// TIA Portal project "2022.05.31_第四章_移动指令3" (V17)

(* hardware
DEVICE "S7-1500/ET200MP station_1"  S7-1500 station
   slot 0: "导轨_0"  Rack  6ES7 590-1***0-0AA0
   slot 1: "PLC_1500"  CPU 1516-3 PN/DP  6ES7 516-3AN00-0AB0  V1.7
      slot 3: "CPU 显示_1"  6ES7591-1BA00-0AA0
      slot 32768: "PROFINET 接口_1"  X1
         slot 32769: "端口_1"  X1 P1
         slot 32770: "端口_2"  X1 P2
      slot 33024: "PROFINET 接口_2"  X2
         slot 33025: "端口_1"  X2 P1
      slot 33280: "DP 接口_1"  X3
DEVICE "HMI_1"  TP1200 Comfort
   slot 0: "HMI_1"  TP1200 Comfort  6AV2 124-0MC01-0AX0  17.0.0.0
   slot 1: "HMI_RT_1"  TP1200 Comfort  6AV2 124-0MC01-0AX0  17.0.0.0
   slot 5: "HMI_1.IE_CP_1"  PROFINET Interface  17.0.0.0
      slot 1: "PROFINET Interface_1"  PROFINET Interface
         slot 1: "Port_1"  Port
         slot 2: "Port_2"  Port
   slot 7: "HMI_1.MPI/DP_CP_1"  MPI/DP Interface  17.0.0.0
*)

// ===== PLC "PLC_1500"  CPU 1516-3 PN/DP =====

DATA_BLOCK "DATE_AND_TIME"   // DB1
{ S7_Optimized_Access := 'TRUE' }
VERSION : 0.1
   VAR
      "time" : Date_And_Time;
      time_ret : Int;
   END_VAR
BEGIN
END_DATA_BLOCK

DATA_BLOCK "启动操作DB"   // DB3
{ S7_Optimized_Access := 'TRUE' }
VERSION : 0.1
   VAR
      从数据数据块中读取按钮 : Bool;
      RET_VAL : Word;
      VALUE : Int;
      写入Array数据块 : Struct
         写入 : Bool;
         按钮 : Bool;
         RET_VAl : Word;
         VALUE : Int;
         写入装载存储器Array数据读取 : Struct
            按钮 : Bool;
            开始读取 : Bool;
            BUSY : Bool;
            DONE : Bool;
            error : Word;
            VALUE : Int;
            写入 : Bool;
            从装载存储器读取Array数据块 : Struct
               按钮 : Bool;
               读取 : Bool;
               BUSY : Bool;
               value : Int;
               done : Bool;
               error : Word;
            END_STRUCT;
         END_STRUCT;
      END_STRUCT;
   END_VAR
BEGIN
END_DATA_BLOCK

DATA_BLOCK "数组数据块A"   // DB4
{ S7_Optimized_Access := 'TRUE' }
VERSION : 0.1
   VAR
      Header : ArrayDBHeader;
      THIS : Array[0..10] of Int;
   END_VAR
BEGIN
END_DATA_BLOCK

DATA_BLOCK "装载数据块"   // DB5
{ S7_Optimized_Access := 'TRUE' }
VERSION : 0.1
BEGIN
END_DATA_BLOCK

FUNCTION_BLOCK "移动指令"   // FB1, LAD
{ S7_Optimized_Access := 'TRUE' }
VERSION : 0.1
   VAR
      ReadFromArrayDBL_Instance : ReadFromArrayDBL;
      WriteToArrayDBL_Instance : WriteToArrayDBL;
      IEC_Timer_0_Instance : TON_TIME;
   END_VAR
   VAR_TEMP   // added for the SCL form of the ladder/FBD networks
      _w1 : Bool;
   END_VAR
BEGIN

REGION Network 1: 从装载存储器Array的数据模块
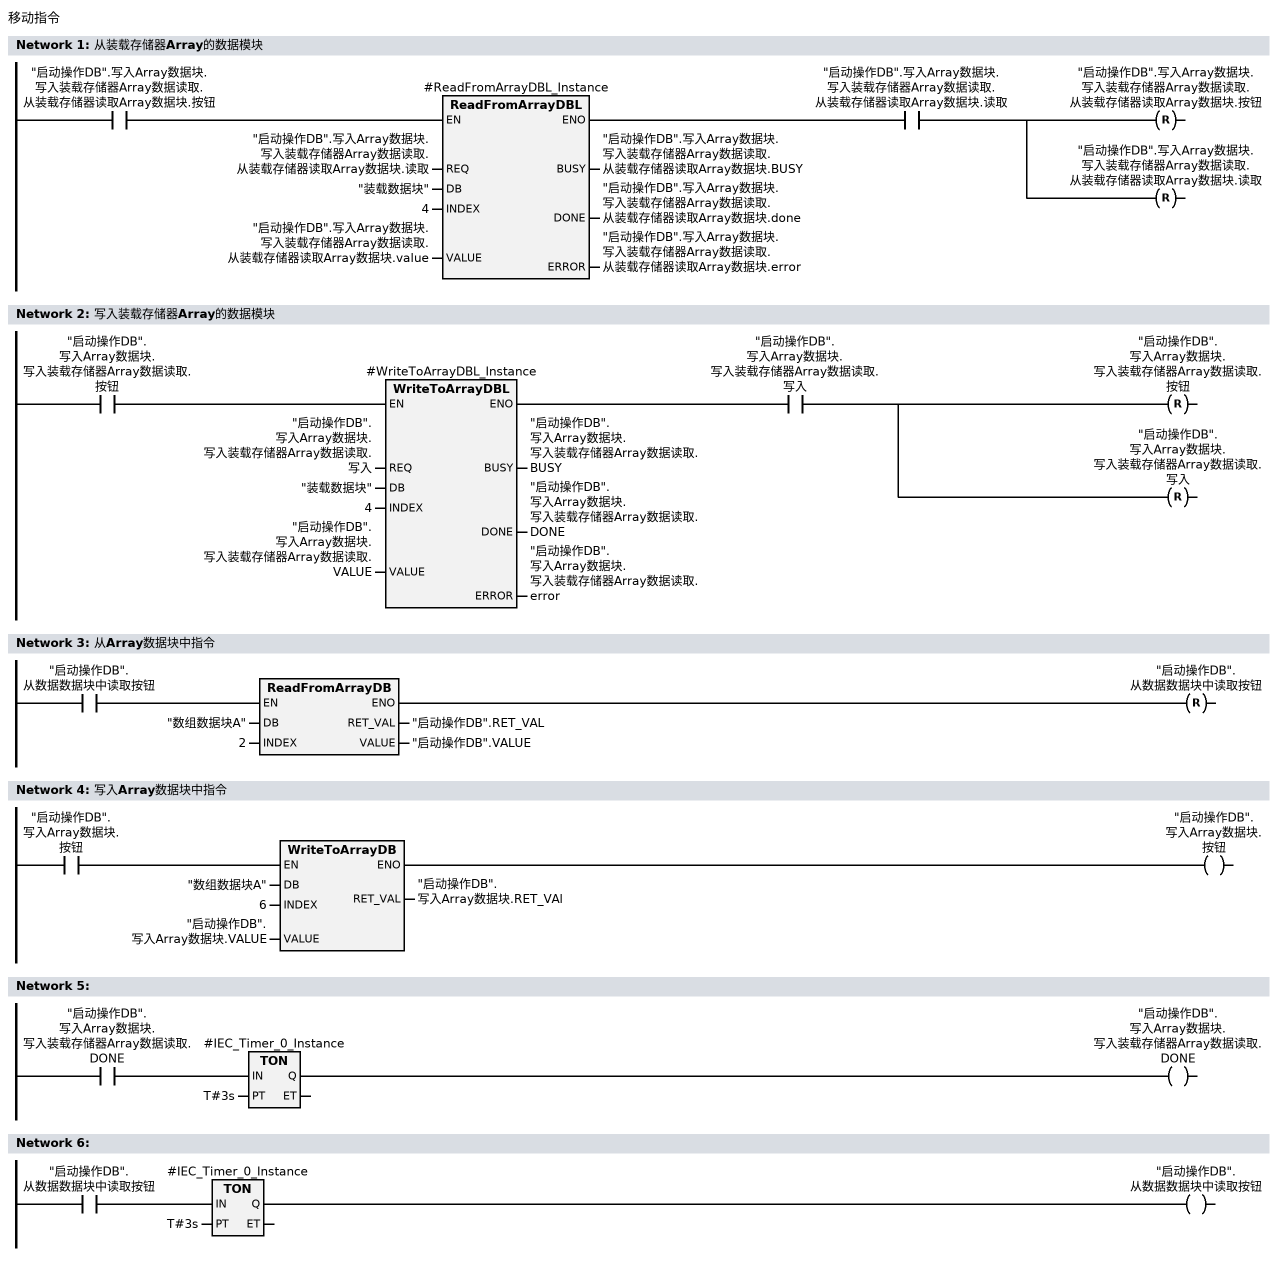
   // ENO of a box is taken as its EN; it also drops when the box reports an error
   #_w1 := "启动操作DB".写入Array数据块.写入装载存储器Array数据读取.从装载存储器读取Array数据块.按钮;
   IF #_w1 THEN
       #ReadFromArrayDBL_Instance(req := "启动操作DB".写入Array数据块.写入装载存储器Array数据读取.从装载存储器读取Array数据块.读取,   // ReadFromArrayDBL
                               db := "装载数据块",
                               index := 4,
                               value := "启动操作DB".写入Array数据块.写入装载存储器Array数据读取.从装载存储器读取Array数据块.value,
                               busy => "启动操作DB".写入Array数据块.写入装载存储器Array数据读取.从装载存储器读取Array数据块.BUSY,
                               done => "启动操作DB".写入Array数据块.写入装载存储器Array数据读取.从装载存储器读取Array数据块.done,
                               error => "启动操作DB".写入Array数据块.写入装载存储器Array数据读取.从装载存储器读取Array数据块.error);
   END_IF;
   IF #_w1 AND "启动操作DB".写入Array数据块.写入装载存储器Array数据读取.从装载存储器读取Array数据块.读取 THEN
       "启动操作DB".写入Array数据块.写入装载存储器Array数据读取.从装载存储器读取Array数据块.按钮 := FALSE;
       "启动操作DB".写入Array数据块.写入装载存储器Array数据读取.从装载存储器读取Array数据块.读取 := FALSE;
   END_IF;
END_REGION

REGION Network 2: 写入装载存储器Array的数据模块
   // ENO of a box is taken as its EN; it also drops when the box reports an error
   #_w1 := "启动操作DB".写入Array数据块.写入装载存储器Array数据读取.按钮;
   IF #_w1 THEN
       #WriteToArrayDBL_Instance(req := "启动操作DB".写入Array数据块.写入装载存储器Array数据读取.写入,   // WriteToArrayDBL
                               db := "装载数据块",
                               index := 4,
                               value := "启动操作DB".写入Array数据块.写入装载存储器Array数据读取.VALUE,
                               busy => "启动操作DB".写入Array数据块.写入装载存储器Array数据读取.BUSY,
                               done => "启动操作DB".写入Array数据块.写入装载存储器Array数据读取.DONE,
                               error => "启动操作DB".写入Array数据块.写入装载存储器Array数据读取.error);
   END_IF;
   IF #_w1 AND "启动操作DB".写入Array数据块.写入装载存储器Array数据读取.写入 THEN
       "启动操作DB".写入Array数据块.写入装载存储器Array数据读取.按钮 := FALSE;
       "启动操作DB".写入Array数据块.写入装载存储器Array数据读取.写入 := FALSE;
   END_IF;
END_REGION

REGION Network 3: 从Array数据块中指令
   // no SCL statement known for ReadFromArrayDB: written as a call
   // ENO of a box is taken as its EN; it also drops when the box reports an error
   #_w1 := "启动操作DB".从数据数据块中读取按钮;
   IF #_w1 THEN
       "启动操作DB".RET_VAL := ReadFromArrayDB(db := "数组数据块A", index := 2, value => "启动操作DB".VALUE);
       "启动操作DB".从数据数据块中读取按钮 := FALSE;
   END_IF;
END_REGION

REGION Network 4: 写入Array数据块中指令
   // no SCL statement known for WriteToArrayDB: written as a call
   // ENO of a box is taken as its EN; it also drops when the box reports an error
   #_w1 := "启动操作DB".写入Array数据块.按钮;
   IF #_w1 THEN
       "启动操作DB".写入Array数据块.RET_VAl := WriteToArrayDB(db := "数组数据块A", index := 6, value := "启动操作DB".写入Array数据块.VALUE);
   END_IF;
   "启动操作DB".写入Array数据块.按钮 := #_w1;
END_REGION

REGION Network 5
   #IEC_Timer_0_Instance(IN := "启动操作DB".写入Array数据块.写入装载存储器Array数据读取.DONE, PT := T#3s);   // TON
   "启动操作DB".写入Array数据块.写入装载存储器Array数据读取.DONE := #IEC_Timer_0_Instance.Q;
END_REGION

REGION Network 6
   #IEC_Timer_0_Instance(IN := "启动操作DB".从数据数据块中读取按钮, PT := T#3s);   // TON
   "启动操作DB".从数据数据块中读取按钮 := #IEC_Timer_0_Instance.Q;
END_REGION
END_FUNCTION_BLOCK

ORGANIZATION_BLOCK "Main"   // OB1, LAD, ProgramCycle
TITLE = "Main Program Sweep (Cycle)"
{ S7_Optimized_Access := 'TRUE' }
VERSION : 0.1
   VAR_INPUT
      Initial_Call : Bool;   // Initial call of this OB
      Remanence : Bool;   // =True, if remanent data are available
   END_VAR
BEGIN

REGION Network 1
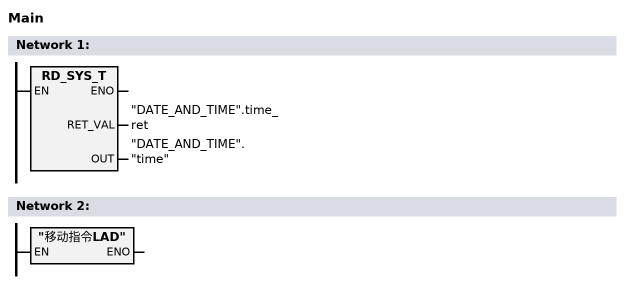
   "DATE_AND_TIME".time_ret := RD_SYS_T(OUT => "DATE_AND_TIME"."time");
END_REGION

REGION Network 2
   RUNG wire#powerrail
      "移动指令LAD"()
   END_RUNG
   // the same network as SCL:
   "移动指令LAD"();
END_REGION
END_ORGANIZATION_BLOCK

(* ===== HMI "HMI_RT_1" =====
system functions are stored by id; their names below are inferred from use
connection "PLC_1500": ETHERNET, S7_1500_OMS
connection "Connection_1": ETHERNET, S7_1500_OMS

HMI tags "默认变量表"
   "DATE_AND_TIME_time_ret" : Int = PLC "DATE_AND_TIME".time_ret, 1 s
   "启动操作DB_从数据数据块中读取按钮" : Bool = PLC 启动操作DB.从数据数据块中读取按钮, 1 s
   "启动操作DB_写入Array数据块_按钮" : Bool = PLC 启动操作DB.写入Array数据块.按钮, 1 s
   "启动操作DB_写入Array数据块_VALUE" : Int = PLC 启动操作DB.写入Array数据块.VALUE, 1 s
   "数组数据块A_THIS{6}" : Int = PLC 数组数据块A.THIS[6], 1 s
   "启动操作DB_写入Array数据块_写入装载存储器Array数据读取_按钮" : Bool = PLC 启动操作DB.写入Array数据块.写入装载存储器Array数据读取.按钮, 1 s
   "启动操作DB_写入Array数据块_写入装载存储器Array数据读取_开始读取" : Bool = PLC 启动操作DB.写入Array数据块.写入装载存储器Array数据读取.开始读取, 1 s
   "启动操作DB_写入Array数据块_写入" : Bool = PLC 启动操作DB.写入Array数据块.写入, 1 s
   "启动操作DB_写入Array数据块_写入装载存储器Array数据读取_写入" : Bool = PLC 启动操作DB.写入Array数据块.写入装载存储器Array数据读取.写入, 1 s
   "启动操作DB_写入Array数据块_写入装载存储器Array数据读取_从装载存储器Array数据块_读取" : Bool = PLC 启动操作DB.写入Array数据块.写入装载存储器Array数据读取.从装载存储器读取Array数据块.读取, 1 s
   "启动操作DB_写入Array数据块_写入装载存储器Array数据读取_从装载存储器Array数据块_done" : Bool = PLC 启动操作DB.写入Array数据块.写入装载存储器Array数据读取.从装载存储器读取Array数据块.done, 1 s
   "启动操作DB_写入Array数据块_写入装载存储器Array数据读取_DONE" : Bool = PLC 启动操作DB.写入Array数据块.写入装载存储器Array数据读取.DONE, 1 s

HMI tags "外部变量"
   "DATE_AND_TIME_time" : Date_And_Time = PLC "DATE_AND_TIME".time, 1 s

HMI tags "内部变量"
   "画面切换颜色" : Int, internal

screen "首页" 1280x740, template "模板_1"
   on GenerateScreen: SetTag("画面切换颜色", 1)

Template "模板_1" 1280x740
   Button "Template_Button_13" at 81,679 size 153x59; TextOff '用户界面1'
      on Release: ActivateScreen("用户界面1", 0); SetTag("画面切换颜色", 2)
      Appearance <- "画面切换颜色"
   Button "退出" at 1200,679 size 78x59; TextOff '退出'; PictureOff "ExitRuntime_TP1200_Comfort_TR"; PictureOn "ExitRuntime_TP1200_Comfort_TR"
      on Release: StopRuntime(0)
   Button "起始画面" at 1,679 size 78x59; TextOff '起始画面'; PictureOff "NavigateHome_TP1200_Comfort_TR"; PictureOn "NavigateHome_TP1200_Comfort_TR"
      on Release: SetTag("画面切换颜色", 1); ActivateScreen("首页", 0)
      Appearance <- "画面切换颜色"
   Button "Template_Button_1" at 236,679 size 153x59; TextOn '用户界面2'; TextOff '用户界面2'
      on Release: ActivateScreen("用户界面2", 0); SetTag("画面切换颜色", 3)
      Appearance <- "画面切换颜色"
   Button "Template_Button_2" at 393,678 size 153x59; TextOn '测试界面'; TextOff '测试界面'
      on Release: ActivateScreen("测试界面", 0); SetTag("画面切换颜色", 4)
      Appearance <- "画面切换颜色"
   Button "Template_Button_3" at 551,678 size 153x59; TextOn '用户管理界面'; TextOff '用户管理界面'
      on Release: ActivateScreen("用户管理界面", 0); SetTag("画面切换颜色", 5)
      Appearance <- "画面切换颜色"
   Button "Template_Button_4" at 710,678 size 153x59; TextOn '报警管理界面'; TextOff '报警管理界面'
      on Release: ActivateScreen("报警视图画面", 0); SetTag("画面切换颜色", 6)
      Appearance <- "画面切换颜色"
   Button "Template_Button_5" at 868,678 size 153x59; TextOn '系统诊断界面'; TextOff '系统诊断界面'
      on Release: ActivateScreen("系统诊断界面", 0); SetTag("画面切换颜色", 7)
      Appearance <- "画面切换颜色"
   Button "Template_Button_6" at 1027,678 size 153x59; TextOn '备用界面'; TextOff '备用界面'
      on Release: ActivateScreen("备用界面", 0); SetTag("画面切换颜色", 8)
      Appearance <- "画面切换颜色"

screen "用户界面1" 1280x740, template "模板_1"
   IOField "I/O 域_1" at 126,102 size 96x32; FormatPattern 9999999
   Button "按钮_1" at 280,102 size 96x32; TextOff '移动'
      on Press: SetBit("启动操作DB_从数据数据块中读取按钮")
   IOField "I/O 域_2" at 437,102 size 96x32; FormatPattern 9999999
   TextField "文本域_1" at 235,57 size 217x21; Text '从Array数据块中读取指令'
   Button "按钮_2" at 280,313 size 96x32; TextOff '移动'
      on Press: SetBit("启动操作DB_从数据数据块中读取按钮")
      on Click: SetBit("启动操作DB_写入Array数据块_按钮")
   TextField "文本域_2" at 235,268 size 199x21; Text '写入Array数据块中指令'
   IOField "I/O 域_3" at 126,313 size 96x32; FormatPattern s99999
      ProcessValue <- "启动操作DB_写入Array数据块_VALUE"
   IOField "I/O 域_4" at 443,313 size 96x32; FormatPattern s99999
      ProcessValue <- "数组数据块A_THIS{6}"
   Button "按钮_3" at 700,205 size 96x44; TextOff '移动'
      on Click: SetBit("启动操作DB_写入Array数据块_写入装载存储器Array数据读取_按钮")
      on Press: SetBit("启动操作DB_从数据数据块中读取按钮")
   TextField "文本域_3" at 757,89 size 235x21; Text '写入装载存储器Array数据块'
   IOField "I/O 域_5" at 796,134 size 96x44; FormatPattern s99999
      ProcessValue <- "启动操作DB_写入Array数据块_VALUE"
   Button "按钮_4" at 896,205 size 96x44; TextOff '写入'
      on Click: SetBit("启动操作DB_写入Array数据块_写入装载存储器Array数据读取_写入")
      on Press: SetBit("启动操作DB_从数据数据块中读取按钮")
   TextField "文本域_4" at 720,274 size 95x21; Text '写入成功：'
   TextField "文本域_5" at 8,8 size 45x21; Text 'Text'
   TextField "文本域_6" at 689,320 size 275x21; Text '住：必须先按移动按钮，再按写入'
   TextField "文本域_7" at 749,375 size 271x21; Text '从装载存储器Array数据块中读取'
   Button "按钮_5" at 700,419 size 96x44; TextOff '移动'
      on Click: SetBit("启动操作DB_写入Array数据块_写入装载存储器Array数据读取_按钮")
      on Press: SetBit("启动操作DB_从数据数据块中读取按钮")
   Button "按钮_6" at 896,419 size 96x44; TextOff '读取'
      on Click: SetBit("启动操作DB_写入Array数据块_写入装载存储器Array数据读取_写入")
      on Press: SetBit("启动操作DB_写入Array数据块_写入装载存储器Array数据读取_从装载存储器Array数据块_读取")
   IOField "I/O 域_6" at 805,551 size 96x44; FormatPattern s99999
      ProcessValue <- "启动操作DB_写入Array数据块_VALUE"
   TextField "文本域_8" at 722,476 size 95x21; Text '读取成功：'
   Circle "圆_2" at 818,471 size 30x30
      Appearance <- "启动操作DB_写入Array数据块_写入装载存储器Array数据读取_从装载存储器Array数据块_done"
   TextField "文本域_9" at 700,513 size 275x21; Text '住：必须先按移动按钮，再按读取'

screen "用户管理界面" 1280x740, template "模板_1"
   UserView "用户视图_1" at 2,2 size 1277x676

screen "报警视图画面" 1280x740, template "模板_1"
   AlarmView "报警视图_1" at 0,0 size 1280x676

screen "系统诊断界面" 1280x740, template "模板_1"
   SysDiagControl "系统诊断视图_1" at 0,2 size 1278x676
*)